// LS Electric XG5000 project: 아파트
// PLC LSPLC
// module base 0 slot 0: 입출력 모듈:XBC-DR14E (DC 24V 입력 8점, 릴레이 출력 6점)

PROGRAM NewProgram (task: 스캔 프로그램)

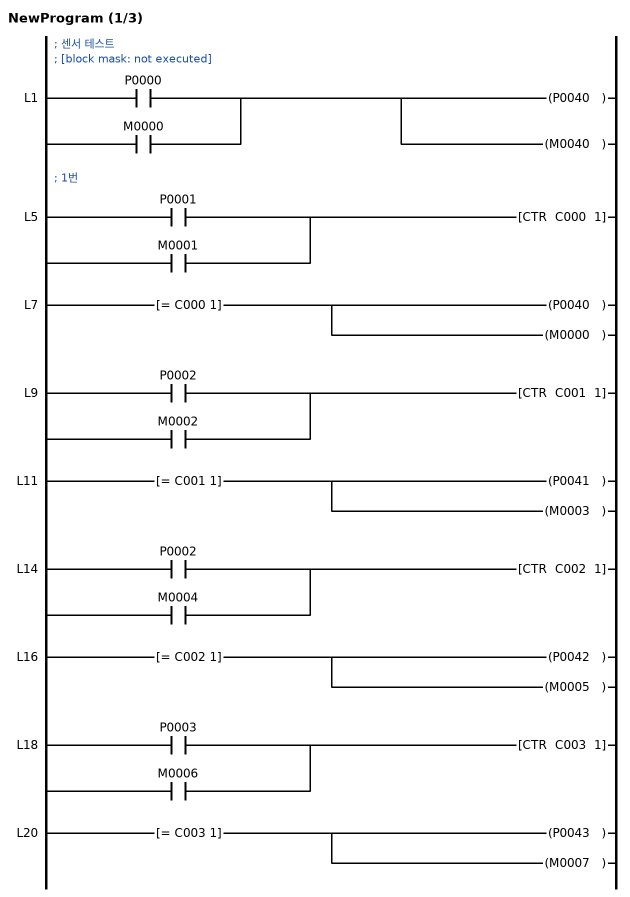
// 센서 테스트
; L1 (block mask: not executed)
LOAD      P0000
OR        M0000
OUT       P0040
OUT       M0040
// 1번
; L5
LOAD      P0001
OR        M0001
CTR       C000 1
; L7
LOAD=     C000 1
OUT       P0040
OUT       M0000
; L9
LOAD      P0002
OR        M0002
CTR       C001 1
; L11
LOAD=     C001 1
OUT       P0041
OUT       M0003
; L14
LOAD      P0002
OR        M0004
CTR       C002 1
; L16
LOAD=     C002 1
OUT       P0042
OUT       M0005
; L18
LOAD      P0003
OR        M0006
CTR       C003 1
; L20
LOAD=     C003 1
OUT       P0043
OUT       M0007

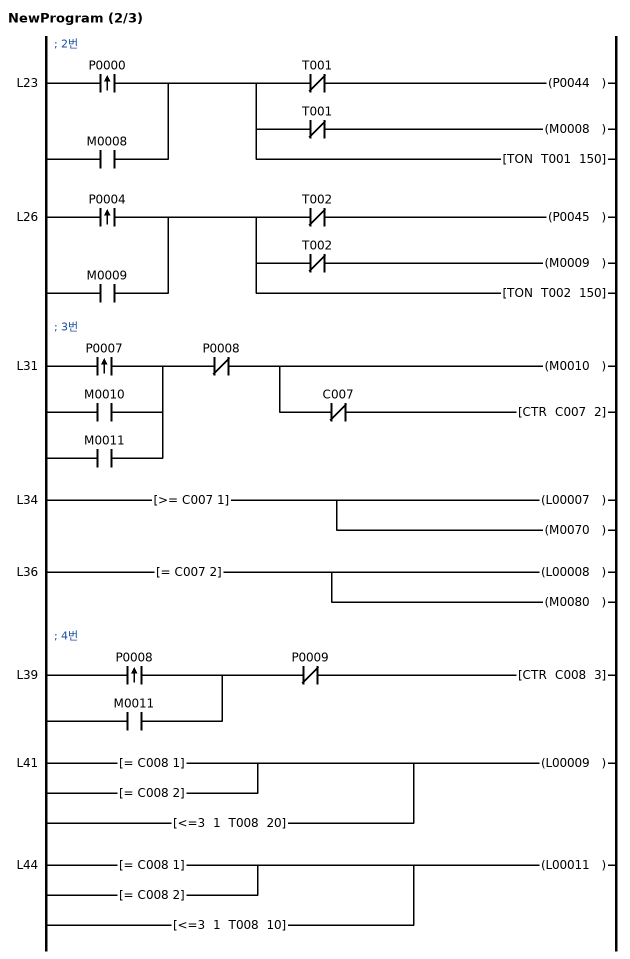
// 2번
; L23
LOADP     P0000
OR        M0008
MPUSH
AND NOT   T001
OUT       P0044
MLOAD
AND NOT   T001
OUT       M0008
MPOP
TON       T001 150
; L26
LOADP     P0004
OR        M0009
MPUSH
AND NOT   T002
OUT       P0045
MLOAD
AND NOT   T002
OUT       M0009
MPOP
TON       T002 150
// 3번
; L31
LOADP     P0007
OR        M0010
OR        M0011
AND NOT   P0008
OUT       M0010
AND NOT   C007
CTR       C007 2
; L34
LOAD>=    C007 1
OUT       L00007
OUT       M0070
; L36
LOAD=     C007 2
OUT       L00008
OUT       M0080
// 4번
; L39
LOADP     P0008
OR        M0011
AND NOT   P0009
CTR       C008 3
; L41
LOAD=     C008 1
OR=       C008 2
OR<=3     1 T008 20
OUT       L00009
; L44
LOAD=     C008 1
OR=       C008 2
OR<=3     1 T008 10
OUT       L00011

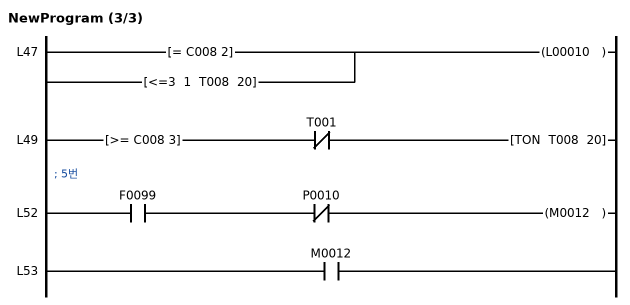
; L47
LOAD=     C008 2
OR<=3     1 T008 20
OUT       L00010
; L49
LOAD>=    C008 3
AND NOT   T001
TON       T008 20
// 5번
; L52
LOAD      F0099
AND NOT   P0010
OUT       M0012
; L53
LOAD      M0012